Universal Robots PolyScope program: 20240827calipoint.urp

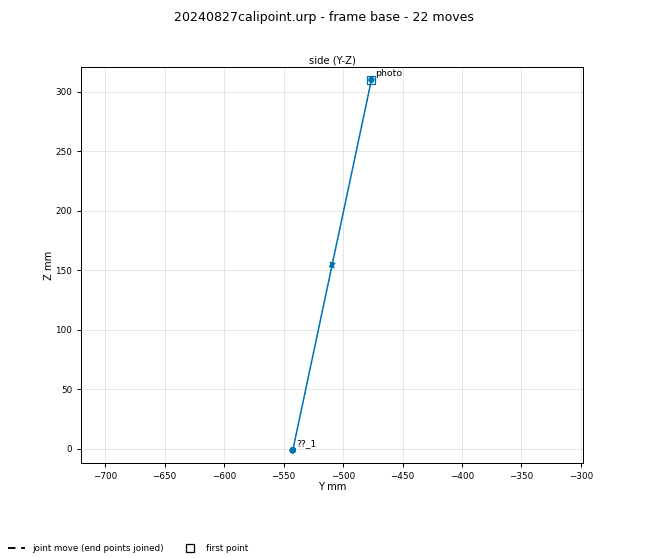
[picture p0: tool path of 20240827calipoint.urp in frame base, 22 of 22 moves have a stored position in this frame; points joined in program order, loops and branches not executed]
Program 20240827calipoint (installation=20240827 directory=/programs/Demos createdIn=5.15.1 lastSavedIn=5.15.1 robotSerialNumber=20245500285)
Calibrated DH parameters: a=[0.000097, -0.210459, -0.026602, 0.000137, 0.000078, 0]; d=[0.162601, 254.180657, -54.076236, -199.970743, 0.099615, 0.099684]; alpha=[1.569796, -0.001455, 0.001957, 1.570525, -1.571561, 0]; deltaTheta=[0, -1.053331, 8.839472, -1.50296, 0.000002, 0]
InitVariablesNode
Robot Program (runOnlyOnce=true)
  cam := rpc_factory("xmlrpc", "http://192.168.1.5:9130/RPC2")
  SuppressedNode
    Script: move = rpc_factory("xmlrpc","http://192.168.1.5:9121/RPC2")
  MoveJ speed 60 deg/s, acceleration 80 deg/s^2 (useActiveTCP=true positionType=JointAngles) feature=Base
    Waypoint photo: TCP in base x=96.736 y=-476.129 z=310.082 mm, rx=-1.9494 ry=-1.8262 rz=-0.6049 rad; joints [85.471, -80.223, 100.083, -75.625, -90.162, 89.442] deg
    Call takephoto
    SuppressedNode
      Halt
  MoveJ speed 60 deg/s, acceleration 80 deg/s^2 (useActiveTCP=true positionType=JointAngles) feature=Base
    Waypoint 路点_1: TCP in base x=93.502 y=-542.216 z=-1.232 mm, rx=2.0515 ry=1.9239 rz=-0.3884 rad; joints [83.107, -101.219, 136.226, -118.224, -88.512, 86.317] deg; TCP offset x=-230 y=0 z=220 mm, rx=0 ry=-0.5236 rz=0 rad
    Call takephoto
    Waypoint 路点_2: TCP in base x=93.498 y=-542.196 z=-1.249 mm, rx=2.0945 ry=2.1206 rz=-0.8133 rad; joints [102.622, -91.538, 130.854, -118.393, -106.595, 108.742] deg
    Call takephoto
    Waypoint 路点_3: TCP in base x=93.497 y=-542.221 z=-1.231 mm, rx=-1.8558 ry=-2.0794 rz=0.6506 rad; joints [107.307, -78.491, 108.14, -87.39, -111.09, 115.326] deg
    Call takephoto
    Waypoint 路点_4: TCP in base x=93.516 y=-542.183 z=-1.265 mm, rx=-1.6771 ry=-2.0001 rz=0.4556 rad; joints [107.665, -67.147, 90.227, -66.333, -111.063, 116.335] deg
    Call takephoto
    Waypoint 路点_5: TCP in base x=93.513 y=-542.22 z=-1.238 mm, rx=-1.4778 ry=-2.0355 rz=-0.0838 rad; joints [100.322, -51.316, 61.762, -38.652, -109.031, 99.365] deg
    Call takephoto
    Waypoint 路点_6: TCP in base x=93.49 y=-542.201 z=-1.233 mm, rx=-1.4784 ry=-2.2489 rz=-0.4593 rad; joints [90.448, -52.036, 60.302, -39.571, -107.613, 76.395] deg
    Call takephoto
    Waypoint 路点_7: TCP in base x=93.511 y=-542.224 z=-1.237 mm, rx=-1.5023 ry=-2.5145 rz=-0.7186 rad; joints [80.596, -56.713, 68.905, -49.954, -105.109, 54.242] deg
    Call takephoto
    Waypoint 路点_8: TCP in base x=93.521 y=-542.225 z=-1.245 mm, rx=-1.4688 ry=-2.5345 rz=-1.0803 rad; joints [75.605, -46.806, 58.042, -41.311, -102.981, 43.385] deg
    Call takephoto
    Waypoint 路点_9: TCP in base x=93.506 y=-542.218 z=-1.223 mm, rx=1.3734 ry=2.5248 rz=0.9242 rad; joints [72.33, -55.198, 71.88, -55.244, -101.614, 35.398] deg
    Call takephoto
    Waypoint 路点_10: TCP in base x=93.518 y=-542.202 z=-1.241 mm, rx=1.3195 ry=2.6302 rz=0.3093 rad; joints [72.862, -77.948, 102.015, -86.745, -102.441, 35.245] deg
    Call takephoto
    Waypoint 路点_11: TCP in base x=93.506 y=-542.224 z=-1.232 mm, rx=1.1982 ry=2.4808 rz=0.0416 rad; joints [64.892, -87.514, 120.615, -108.822, -95.123, 24.358] deg
    Call takephoto
    Waypoint 路点_12: TCP in base x=93.511 y=-542.189 z=-1.268 mm, rx=1.2179 ry=2.6519 rz=-0.1972 rad; joints [73.708, -92.973, 124.801, -114.657, -103.893, 34.538] deg
    Call takephoto
    Waypoint 路点_13: TCP in base x=93.506 y=-542.184 z=-1.265 mm, rx=1.2254 ry=2.8429 rz=-0.5033 rad; joints [86.997, -94.797, 127.613, -117.875, -117.184, 49.439] deg
    Call takephoto
    Waypoint 路点_14: TCP in base x=93.506 y=-542.214 z=-1.232 mm, rx=-1.1246 ry=-2.6926 rz=0.4129 rad; joints [95.41, -87.533, 115.743, -99.863, -124.679, 61.895] deg
    Call takephoto
    Waypoint 路点_15: TCP in base x=93.485 y=-542.215 z=-1.228 mm, rx=-1.3405 ry=-2.4295 rz=0.4078 rad; joints [102.072, -79.591, 104.802, -81.387, -121.799, 86.556] deg
    Call takephoto
    Wait Sleep waitTime=1
    Call takephoto
    Waypoint 路点_16: TCP in base x=93.503 y=-542.18 z=-1.251 mm, rx=-1.5242 ry=-2.1637 rz=0.2501 rad; joints [103.477, -67.132, 86.573, -61.525, -113.541, 101.599] deg
    Call takephoto
    Waypoint 路点_17: TCP in base x=93.509 y=-542.198 z=-1.238 mm, rx=-2.0144 ry=-1.8049 rz=0.0543 rad; joints [97.848, -62.284, 77.179, -56.247, -95.18, 112.361] deg
    Call takephoto
    Waypoint 路点_18: TCP in base x=93.515 y=-542.191 z=-1.243 mm, rx=-2.1605 ry=-1.5091 rz=-0.1244 rad; joints [94.447, -53.665, 63.988, -46.018, -85.4, 118.38] deg
    Call takephoto
    Waypoint 路点_19: TCP in base x=93.514 y=-542.214 z=-1.242 mm, rx=-2.4315 ry=-1.3166 rz=-0.5223 rad; joints [82.915, -56.191, 66.714, -44.37, -72.542, 108.811] deg
    Call takephoto
    Waypoint 路点_20: TCP in base x=93.495 y=-542.232 z=-1.216 mm, rx=-2.2919 ry=-1.8202 rz=-0.5743 rad; joints [80.06, -63.302, 76.7, -50.399, -82.453, 87.694] deg
    Call takephoto
  MoveJ speed 60 deg/s, acceleration 80 deg/s^2 (useActiveTCP=true positionType=JointAngles) feature=Base
    Waypoint photo: TCP in base x=96.736 y=-476.129 z=310.082 mm, rx=-1.9494 ry=-1.8262 rz=-0.6049 rad; joints [85.471, -80.223, 100.083, -75.625, -90.162, 89.442] deg
SubProgram -> takephoto
SubProgram takephoto (keepSynchronizedWithDisk=false)
  Wait Sleep waitTime=1
  Script: cam.takePhoto(get_actual_tcp_pose())
  Popup Message (haltProgram=false message=please ensure  inputType=Text)
